% RSLogix 500 project Balizas_sensores.RSS, saved by version 8.30.00.16 %
PROJECT "UNTITLED"    % processor: Bul.1763 MicroLogix 1100 Series B %

PROGRAM FILES
  LAD 2   7 rungs

DATA FILES
  O0 OUTPUT  6 elements
  I1 INPUT  12 elements
  S2 STATUS  66 elements
  B3 BINARY  1 elements
  T4 TIMER  1 elements
  C5 COUNTER  1 elements
  R6 CONTROL  1 elements
  N7 INTEGER  2 elements
  F8 FLOAT  3 elements

LADDER 2
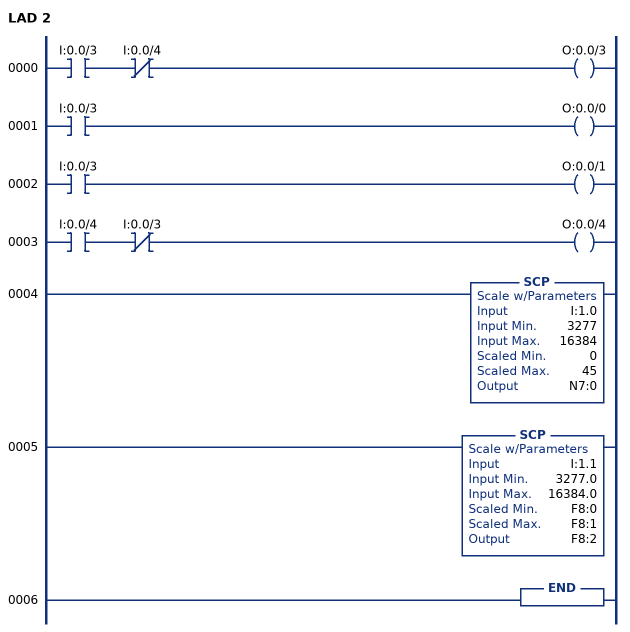
% Rung: 0 %
SOR XIC I:0.0/3 XIO I:0.0/4 OTE O:0.0/3 EOR
% Rung: 1 %
SOR XIC I:0.0/3 OTE O:0.0/0 EOR
% Rung: 2 %
SOR XIC I:0.0/3 OTE O:0.0/1 EOR
% Rung: 3 %
SOR XIC I:0.0/4 XIO I:0.0/3 OTE O:0.0/4 EOR
% Rung: 4 %
SOR SCP I:1.0 3277 16384 0 45 N7:0 EOR
% Rung: 5 %
SOR SCP I:1.1 3277.0 16384.0 F8:0 F8:1 F8:2 EOR
% Rung: 6 %
SOR END EOR

DATA TABLE (non-zero values as saved)
DATA N7
% N7:0 % 36 1
DATA F8
% F8:0 % 3 200 24.1474
